// SIMATIC S7-200 project (STEP 7-Micro/WIN), CPU 224XP REL 02.01

SYMBOL_TABLE USUARIO1
P_TICKET         I0.0
C_FOTOELECTRICA  I0.1
SALIDA_P_BOTONERA I0.2
SALIDA_C_FOTOELECTRICA I0.3
E_SUBIR_BARRERA_ Q0.0
E_BAJAR_BARRERA_ Q0.1
VERDE_LIBRE      Q0.2
ROJO_LLENO       Q0.3
S_SUBIR_BARRERA  Q0.4
S_BAJAR_BARRERA  Q0.5
CONTADOR         MW4
END_SYMBOL_TABLE

ORGANIZATION_BLOCK PRINCIPAL:OB1
TITLE=COMENTARIOS DEL PROGRAMA
BEGIN
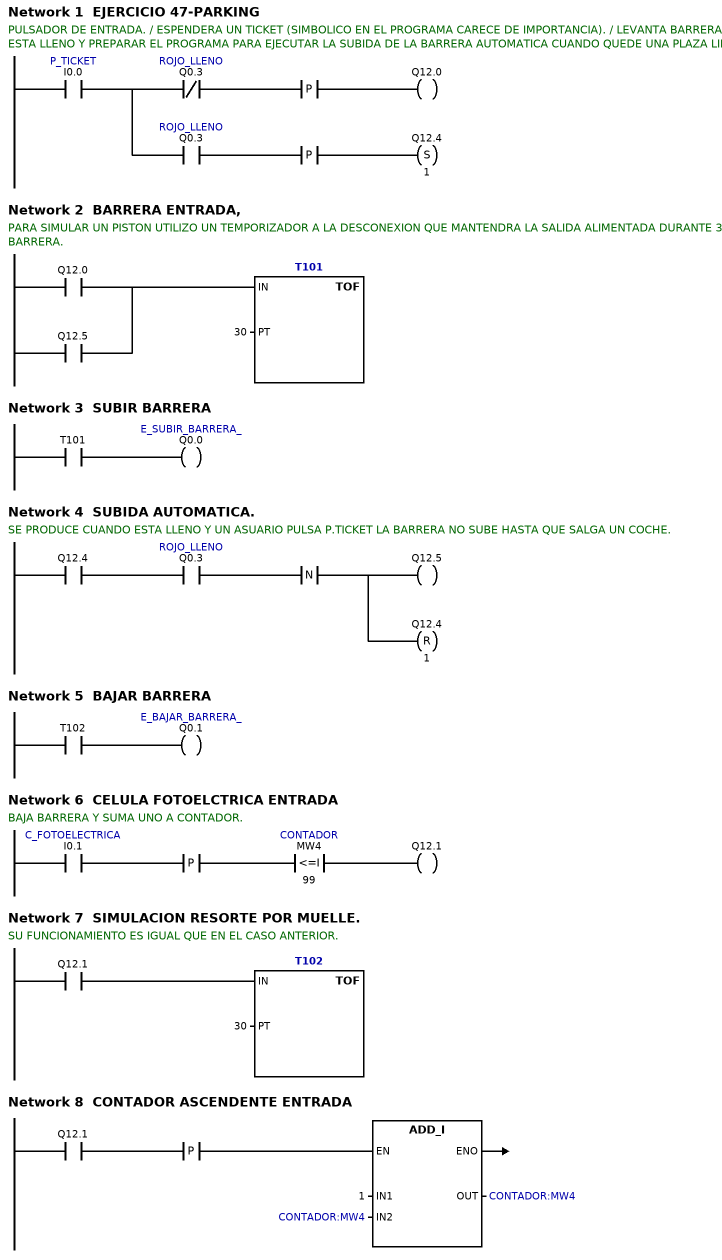
Network 1 // EJERCICIO 47-PARKING
// PULSADOR DE ENTRADA.
// ESPENDERA UN TICKET (SIMBOLICO EN EL PROGRAMA CARECE DE IMPORTANCIA).
// LEVANTA BARRERA.
// MANIOBRA Q12.4 SE ENCARGA DE REGISTRAR EL PULSO CUANDO ESTA LLENO Y PREPARAR EL PROGRAMA PARA EJECUTAR LA SUBIDA DE LA BARRERA AUTOMATICA CUANDO QUEDE UNA PLAZA LIBRE.
LD     P_TICKET:I0.0
LPS
AN     ROJO_LLENO:Q0.3
EU
=      Q12.0
LPP
A      ROJO_LLENO:Q0.3
EU
S      Q12.4, 1
Network 2 // BARRERA ENTRADA,
// PARA SIMULAR UN PISTON UTILIZO UN TEMPORIZADOR A LA DESCONEXION QUE MANTENDRA LA SALIDA ALIMENTADA DURANTE 3 SEG. QUE ES LO QUE TARDA EN EJECUTAR LA ACCION DE SUBIR BARRERA.
LD     Q12.0
O      Q12.5
TOF    T101, 30
Network 3 // SUBIR BARRERA
LD     T101
=      E_SUBIR_BARRERA_:Q0.0
Network 4 // SUBIDA AUTOMATICA.
// SE PRODUCE CUANDO ESTA LLENO Y UN ASUARIO PULSA P.TICKET LA BARRERA NO SUBE HASTA QUE SALGA UN COCHE.
LD     Q12.4
A      ROJO_LLENO:Q0.3
ED
=      Q12.5
R      Q12.4, 1
Network 5 // BAJAR BARRERA
LD     T102
=      E_BAJAR_BARRERA_:Q0.1
Network 6 // CELULA FOTOELCTRICA ENTRADA
// BAJA BARRERA Y SUMA UNO A CONTADOR.
LD     C_FOTOELECTRICA:I0.1
EU
AW<=   CONTADOR:MW4, 99
=      Q12.1
Network 7 // SIMULACION RESORTE POR MUELLE.
// SU FUNCIONAMIENTO ES IGUAL QUE EN EL CASO ANTERIOR.
LD     Q12.1
TOF    T102, 30
Network 8 // CONTADOR ASCENDENTE ENTRADA
LD     Q12.1
EU
+I     1, CONTADOR:MW4
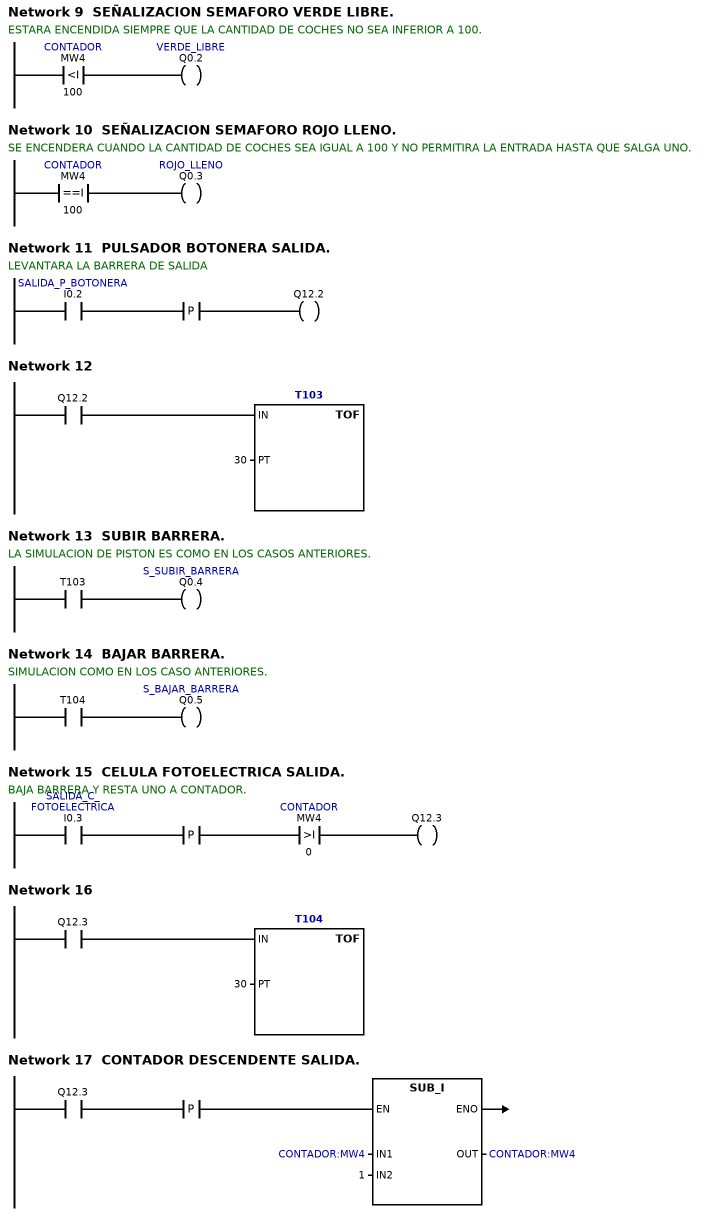
Network 9 // SEÑALIZACION SEMAFORO VERDE LIBRE.
// ESTARA ENCENDIDA SIEMPRE QUE LA CANTIDAD DE COCHES NO SEA INFERIOR A 100.
LDW<   CONTADOR:MW4, 100
=      VERDE_LIBRE:Q0.2
Network 10 // SEÑALIZACION SEMAFORO ROJO LLENO.
// SE ENCENDERA CUANDO LA CANTIDAD DE COCHES SEA IGUAL A 100 Y NO PERMITIRA LA ENTRADA HASTA QUE SALGA UNO.
LDW=   CONTADOR:MW4, 100
=      ROJO_LLENO:Q0.3
Network 11 // PULSADOR BOTONERA SALIDA.
// LEVANTARA LA BARRERA DE SALIDA
LD     SALIDA_P_BOTONERA:I0.2
EU
=      Q12.2
Network 12
LD     Q12.2
TOF    T103, 30
Network 13 // SUBIR BARRERA.
// LA SIMULACION DE PISTON ES COMO EN LOS CASOS ANTERIORES.
LD     T103
=      S_SUBIR_BARRERA:Q0.4
Network 14 // BAJAR BARRERA.
// SIMULACION COMO EN LOS CASO ANTERIORES.
LD     T104
=      S_BAJAR_BARRERA:Q0.5
Network 15 // CELULA FOTOELECTRICA SALIDA.
// BAJA BARRERA Y RESTA UNO A CONTADOR.
LD     SALIDA_C_FOTOELECTRICA:I0.3
EU
AW>    CONTADOR:MW4, 0
=      Q12.3
Network 16
LD     Q12.3
TOF    T104, 30
Network 17 // CONTADOR DESCENDENTE SALIDA.
LD     Q12.3
EU
-I     1, CONTADOR:MW4
END_ORGANIZATION_BLOCK
